FUNCTION_BLOCK FB_Example
VAR
    iValue : INT;
END_VAR
BEGIN
iValue := 5
END_FUNCTION_BLOCK
